// TIA Portal V19 export
TYPE "SmartLoopControl_Par"
// stored: Access Published
   STRUCT
      WorkMode { S7_SetPoint := 'True'} : UInt;   // 0 = Sensors; 1 =Material counters
      SyncEntryMode { S7_SetPoint := 'True'} : UInt;   // 0=Reduce;1=Stop
      SyncExitMode { S7_SetPoint := 'True'} : UInt;   // 0=Reduce;1=Stop
      PosStopMinHigh { S7_SetPoint := 'True'} : LReal;
      PosStopMiddle { S7_SetPoint := 'True'} : LReal;
      PosStopMaxLow { S7_SetPoint := 'True'} : LReal;
      PosSynch { S7_SetPoint := 'True'} : LReal;
      PosDeltaRestartAfterMaxLow { S7_SetPoint := 'True'} : LReal;
      PosDeltaRestartAfteMinHigh { S7_SetPoint := 'True'} : LReal;
      PosIntervalSynchroCyclic { S7_SetPoint := 'True'} : LReal;
      HysteresysSynchroExt { S7_SetPoint := 'True'} : LReal;
      Entry_Lim1_VMin { S7_SetPoint := 'True'} : LReal;
      Entry_Lim2_VMed { S7_SetPoint := 'True'} : LReal;
      Entry_Lim3_VMax { S7_SetPoint := 'True'} : LReal;
      Entry_Override1_VMin { S7_SetPoint := 'True'} : LReal;
      Entry_Override2_VMed { S7_SetPoint := 'True'} : LReal;
      Entry_Override3_VMax { S7_SetPoint := 'True'} : LReal;
      Exit_Lim1_VMin { S7_SetPoint := 'True'} : LReal;
      Exit_Lim2_VMed { S7_SetPoint := 'True'} : LReal;
      Exit_Lim3_VMax { S7_SetPoint := 'True'} : LReal;
      Exit_Override1_VMin { S7_SetPoint := 'True'} : LReal;
      Exit_Override2_VMed { S7_SetPoint := 'True'} : LReal;
      Exit_Override3_VMax { S7_SetPoint := 'True'} : LReal;
      DlySetMaxLow { S7_SetPoint := 'True'} : Time;
      DlyRstMaxLow { S7_SetPoint := 'True'} : Time;
      Exit_MaxFeed_CaseSystemOff { S7_SetPoint := 'True'} : LReal;
      Exit_MaxFeed_CaseNextEndOfMaterial { S7_SetPoint := 'True'} : LReal;
      Exit_MaxFeed_CaseLoopMaterialNotValid { S7_SetPoint := 'True'} : LReal;
   END_STRUCT;
END_TYPE
